FUNCTION calcTravelTime : INT
VAR_INPUT
    distance : INT; // in kilometers
    speed : INT;    // in km/h
END_VAR

// Simpele berekening reistijd in minuten
calcTravelTime := (distance) / speed;

END_FUNCTION

(* stored: Version 1.1.0.1, ProductVersion 3.1.4024.15
   POU calcTravelTime: Id {55fc3503-48a6-4b54-aaa0-4cfced1a0548}, SpecialFunc None *)
